// Brief: Slave Arm Init
FUNCTION_BLOCK PUBLIC FB_SlaveCtrlInit EXTENDS FB_SlaveArmCtrlBase
VAR_INPUT
END_VAR
VAR_OUTPUT
END_VAR
VAR
	m_initState :INT :=0;
END_VAR

// override this function in each exact controller
METHOD PROTECTED calcCmdJntPos : BOOL
VAR_IN_OUT CONSTANT
	i_endoscopePose : ST_Frame;
	i_masterStatus :ST_MasterStatus;
	i_setupStatus: ST_SetupStatus;
	i_slaveArm :FB_SlaveArm;
END_VAR

VAR 
	curInstruDepth:LREAL;
END_VAR
IF m_timePeriod > 1.0 THEN
	m_isFinished := true;
END_IF
END_METHOD

METHOD PUBLIC init : BOOL
VAR_IN_OUT CONSTANT
	i_slaveArm	:FB_SlaveArm;
END_VAR
VAR_IN_OUT 
	r_slaveArmCtrlCmd :ST_SlaveArmCtrlCmds;
END_VAR

VAR
	i:INT;
END_VAR
SUPER^.Init(i_slaveArm,r_slaveArmCtrlCmd);
m_jntEnableFlag:=g_zeroVec8i;

// update commands to arm
copyCmds(r_slaveArmCtrlCmd);
END_METHOD

END_FUNCTION_BLOCK

(* stored: Version 1.1.0.1, ProductVersion 3.1.4024.11
   POU FB_SlaveCtrlInit: Id {2f1b91d8-ebd5-4b63-92d8-450fe3a94973}, SpecialFunc None
   Method calcCmdJntPos: Id {50167c08-0683-4e04-ab32-64d931dad4e1}
   Method init: Id {0eca198b-2030-4cc0-a250-a6bdc9d0e230} *)
